{attribute addProperty BoxType "KL1012"}
{attribute addProperty Id "Channel_1Channel_70B606D100Channel_2Channel_70B606D100"}
{attribute addProperty CRC "3525945802"}
{attribute addProperty SizeInBites "0"}
{attribute addProperty SizeInBytes "0"}
TYPE KL1012_D229A9CA :
STRUCT
	{attribute addProperty Name "Channel_1"}
	Channel_1 : Channel_70B606D1;
	{attribute addProperty Name "Channel_2"}
	Channel_2 : Channel_70B606D1;
END_STRUCT
END_TYPE

(* stored: Version 1.2.0.0, ProductVersion 3.1.4024.9
   DUT KL1012_D229A9CA: Id {b0119dd4-5cd4-40a6-bf15-2461e663e916} *)
